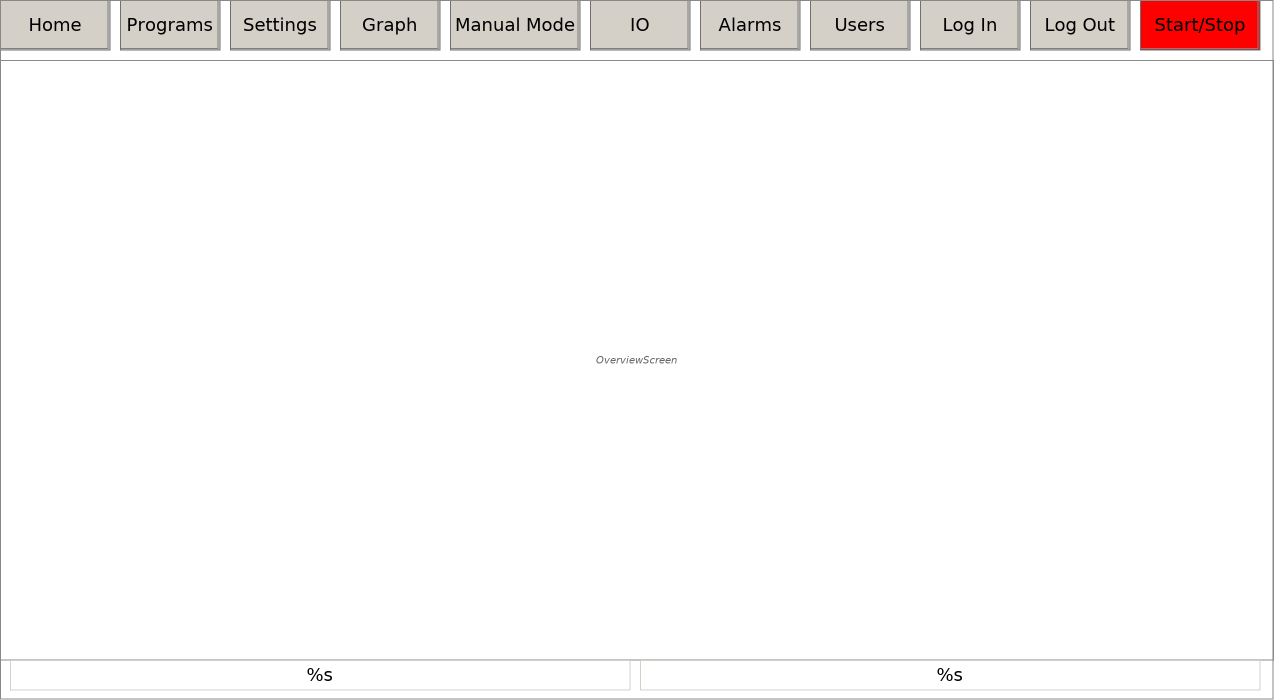
VISUALIZATION HMI_MAIN  // 1274x700
    Button (120,0 100x50), "Programs"
        OnMouseClick: FrameSelectionChange Selection=SelectedFrame=12e04cd0-f39d-4869-84a5-022adc51170e, Selection=1, GlobSel=AssignType=Directly, SelType=Locally
    Frame (0,60 1274x600)
        shows OverviewScreen()
        shows ProgramScreen()
        shows Settings()
        shows GraphScreen()
        shows ManualMode()
        shows IO()
        shows Alarms()
    Button (0,0 110x50), "Home"
        OnMouseClick: FrameSelectionChange Selection=SelectedFrame=12e04cd0-f39d-4869-84a5-022adc51170e, GlobSel=AssignType=Directly, SelType=Locally
    Button (230,0 100x50), "Settings"
        OnMouseClick: FrameSelectionChange Selection=SelectedFrame=12e04cd0-f39d-4869-84a5-022adc51170e, Selection=2, GlobSel=AssignType=Directly, SelType=Locally
    Button (340,0 100x50), "Graph"
        OnMouseClick: FrameSelectionChange Selection=SelectedFrame=12e04cd0-f39d-4869-84a5-022adc51170e, Selection=3, GlobSel=AssignType=Directly, SelType=Locally
    Button (450,0 130x50), "Manual Mode"
        OnMouseClick: FrameSelectionChange Selection=SelectedFrame=12e04cd0-f39d-4869-84a5-022adc51170e, Selection=4, GlobSel=AssignType=Directly, SelType=Locally
    Button (590,0 100x50), "IO"
        OnMouseClick: FrameSelectionChange Selection=SelectedFrame=12e04cd0-f39d-4869-84a5-022adc51170e, Selection=5, GlobSel=AssignType=Directly, SelType=Locally
    Button (700,0 100x50), "Alarms", colour toggle: GVL.bActiveAlarm
        OnMouseClick: FrameSelectionChange Selection=SelectedFrame=12e04cd0-f39d-4869-84a5-022adc51170e, Selection=6, GlobSel=AssignType=Directly, SelType=Locally
    Textfield (10,660 620x30), "%s", text variable: GVL.sAlarmText
    Textfield (640,660 620x30), "%s", text variable: GVL.sInfoText
    Button (920,0 100x50), "Log In"
        OnMouseClick: VisuUserMgmt Type=Login
    Button (1140,0 120x50), "Start/Stop", colour toggle: GVL.HMIPowerButton, input disabled if: GVL.manualMode
        OnMouseClick: toggle GVL.HMIPowerButton
    Button (810,0 100x50), "Users"
        OnMouseClick: VisuUserMgmt Type=OpenUserConfiguration
    Button (1030,0 100x50), "Log Out"
        OnMouseClick: VisuUserMgmt Type=Logout
END_VISUALIZATION

(* stored: Version 1.1.0.1, ProductVersion 3.1.4022.16
   Visu HMI_MAIN: Id {83561f98-e78a-4de4-8243-2a057e1f5cca} *)
